FUNCTION_BLOCK OrderHandling
VAR_INPUT
	mxEnable: BOOL;
	msOrderfornextAssemblyfromStation: STRING;
	msProductNames: Array[1..9] OF STRING;
	mxAGVAtStation: BOOL;
	mxPalletonAGV: BOOL;
	mxAGVoutofStation: BOOL;
END_VAR
VAR_OUTPUT
	mxErrorCode: INT;
	mxAGVLeave: BOOL;
END_VAR
VAR
	order: INT;
END_VAR

IF mxEnable THEN
	CASE order OF
		0:
			IF msOrderfornextAssemblyfromStation <> '0' THEN
				order:= 10;
			END_IF
		10:
			order:=20;
		20:
			IF msOrderfornextAssemblyfromStation = msProductNames[1] THEN
				order:=30;
			ELSIF msOrderfornextAssemblyfromStation = msProductNames[2] THEN
				order:=30;
			ELSIF msOrderfornextAssemblyfromStation = msProductNames[3] THEN
				order:=30;
			ELSIF msOrderfornextAssemblyfromStation = msProductNames[4] THEN
				order:=30;
			ELSIF msOrderfornextAssemblyfromStation = msProductNames[5] THEN
				order:=30;
			ELSIF msOrderfornextAssemblyfromStation = msProductNames[6] THEN
				order:=30;
			ELSIF msOrderfornextAssemblyfromStation = msProductNames[7] THEN
				order:=30;
			ELSIF msOrderfornextAssemblyfromStation = msProductNames[8] THEN
				order:=30;
			ELSIF msOrderfornextAssemblyfromStation = msProductNames[9] THEN
				order:=30;
			ELSIF msOrderfornextAssemblyfromStation = 'AssembledProduct' THEN
				order:=30;
			ELSIF msOrderfornextAssemblyfromStation = 'InvalidPart' THEN
				order:=30;
			ELSE 
				order:=22;
			END_IF 
		22: // Invalid Product Name
			mxErrorCode:=22;
				IF msOrderfornextAssemblyfromStation = '0' THEN
					mxErrorCode:=0;
					order:= 0;
				END_IF
		30:
			CommData.mxRequestAGV:=TRUE;
			IF mxAGVAtStation THEN
				CommData.mxRequestAGV:=FALSE;
				order:=40;
			END_IF
		40:
			IF mxPalletonAGV THEN
				mxAGVLeave:=TRUE;
				order:=50;
			END_IF
		50:
			IF mxAGVoutofStation THEN
				mxAGVLeave:=FALSE;
				order:=60;
			END_IF
		60:
			IF msOrderfornextAssemblyfromStation = '0' THEN
				order:= 0;
			END_IF
	END_CASE
END_IF

END_FUNCTION_BLOCK

(* stored: Version 1.1.0.1, ProductVersion 3.1.4022.16
   POU OrderHandling: Id {0055eee3-1759-468e-b376-63e0e9a8e98c}, SpecialFunc None *)
